// TIA Portal V15.1 export
// export: Created 2024-05-17T05:38:25.7999474Z, ExportSetting WithDefaults, DisplayName Totally Integrated Automation Portal, DisplayVersion V15.1 Update 5, DisplayName TIA Portal Openness, DisplayVersion V15.1 Update 5, DisplayName SINAMICS Startdrive Advanced, DisplayVersion V15.1, DisplayName G130, G150, S120, S150, SINAMICS MV, S210, DisplayVersion V15.1, DisplayName G110M, G120, G120C, G120D, G120P, DisplayVersion V15.1, DisplayName STEP 7 Professional, DisplayVersion V15.1 Update 5, DisplayName STEP 7 Safety, DisplayVersion V15.1, DisplayName WinCC Professional, DisplayVersion V15.1 Update 5, DisplayName SIMATIC Visualization Architect, DisplayVersion V15.1
FUNCTION "LHmiLed" : Void   // FC1008, FBD
TITLE = LHmiLed
{ S7_Optimized_Access := 'FALSE' }
AUTHOR : VCC
FAMILY : Control
NAME : HmiLed
VERSION : 1.0
// ================================================================================
// This module handles indication for Start, Alarm reset and Cycle stop button.
// ================================================================================
// stored: AutoNumber false, IsIECCheckEnabled false, SetENOAutomatically False, UDAEnableTagReadback false
   VAR_INPUT
      I_AlarmABCondition : Bool;   // Alarm AB condition
      I_AlarmAB : Bool;   // Alarm AB active
      I_AutoMode : Bool;   // Auto mode
      I_AutoSel : Bool;   // Auto selected
      I_CycleStopRequest : Bool;   // Cycle stop request
      I_CycleStopReached : Bool;   // Cycle stop reached
      I_Lamptest : Bool;   // Lamptest
   END_VAR
   VAR_OUTPUT
      O_StartPBInd : Bool;   // Start PB indication
      O_AlarmResetPBInd : Bool;   // Alarm reset PB indicatio
      O_CycleStopPBInd : Bool;   // Cycle stop PB indication
   END_VAR
BEGIN

REGION Network 1: **** 4.6 - Machine Status - Indications **** Alarm reset PB indication
   // Alarm reset PB indication
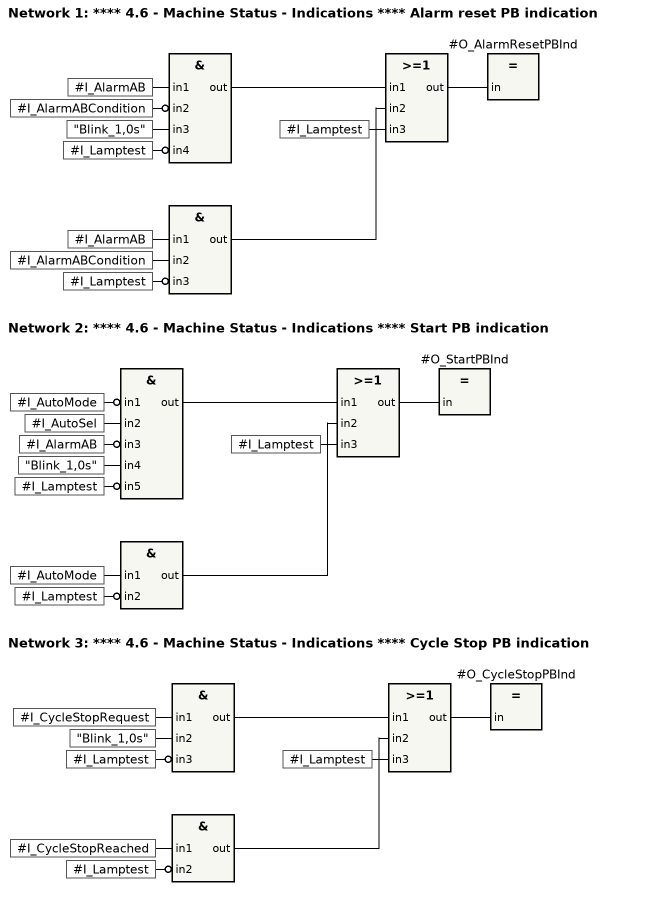
   #O_AlarmResetPBInd := (#I_AlarmAB AND NOT #I_AlarmABCondition AND "Blink_1,0s" AND NOT #I_Lamptest) OR (#I_AlarmAB AND #I_AlarmABCondition AND NOT #I_Lamptest) OR #I_Lamptest;
END_REGION

REGION Network 2: **** 4.6 - Machine Status - Indications **** Start PB indication
   // Start PB indication
   #O_StartPBInd := (NOT #I_AutoMode AND #I_AutoSel AND NOT #I_AlarmAB AND "Blink_1,0s" AND NOT #I_Lamptest) OR (#I_AutoMode AND NOT #I_Lamptest) OR #I_Lamptest;
END_REGION

REGION Network 3: **** 4.6 - Machine Status - Indications **** Cycle Stop PB indication
   // Cycle Stop PB indication
   #O_CycleStopPBInd := (#I_CycleStopRequest AND "Blink_1,0s" AND NOT #I_Lamptest) OR (#I_CycleStopReached AND NOT #I_Lamptest) OR #I_Lamptest;
END_REGION
END_FUNCTION
